Fanuc TP program (LS listing): TEMPLATE.LS

/PROG  TEMPLATE
/ATTR
OWNER		= MNEDITOR;
COMMENT		= "Template for Progs";
PROG_SIZE	= 363;
CREATE		= DATE 21-08-29  TIME 13:28:02;
MODIFIED	= DATE 21-08-29  TIME 13:28:32;
FILE_NAME	= ;
VERSION		= 0;
LINE_COUNT	= 25;
MEMORY_SIZE	= 635;
PROTECT		= READ_WRITE;
TCD:  STACK_SIZE	= 0,
      TASK_PRIORITY	= 50,
      TIME_SLICE	= 0,
      BUSY_LAMP_OFF	= 0,
      ABORT_REQUEST	= 0,
      PAUSE_REQUEST	= 0;
DEFAULT_GROUP	= 1,*,*,*,*;
CONTROL_CODE	= 00000000 00000000;
LOCAL_REGISTERS	= 0,0,0;
/APPL

AUTO_SINGULARITY_HEADER;
  ENABLE_SINGULARITY_AVOIDANCE   : TRUE;
/MN
   1:   !--------------------!;
   2:   !  Program Header;
   3:   !--------------------!;
   4:   ;
   5:   ;
   6:   ;
   7:   ;
   8:   ;
   9:   ;
  10:   !----INFORMATION----;
  11:   ;
  12:   ;
  13:   ;
  14:   ;
  15:   ;
  16:   ;
  17:   ;
  18:   ;
  19:   ;
  20:   ;
  21:   ;
  22:   END;
  23:   !---TOUCH UP AREA----;
  24:   ;
  25:   ;
/POS
/END
